// TwinCAT 3 PLC project plc_application1
// ProgramVersion: 3.1.4022.7
// libraries:
//   Tc2_Standard, * (Beckhoff Automation GmbH)
//   Tc2_System, * (Beckhoff Automation GmbH)
//   Tc3_Module, * (Beckhoff Automation GmbH)
// project tree:
//   DUTs/ DUT_1.TcDUT
//   GVLs/ GVL.TcGVL, GVL_1.TcGVL
//   / PlcTask.TcTTO
//   POUs/ MAIN.TcPOU, POU.TcPOU
// real-time tasks:
//   TASK PlcTask: cycle T#10ms, priority 20, ADS port 350
// I/O:
//   DEVICE Device 1 (EtherCAT), AmsNetId 10.1.1.164.2.1

CONFIGURATION plc_application1
    RESOURCE PLC ON TwinCAT3
        TASK PlcTask(INTERVAL := T#10ms, PRIORITY := 20);
        PROGRAM MAIN WITH PlcTask : MAIN;
    END_RESOURCE
END_CONFIGURATION

// ---- DUTs/DUT_1.TcDUT
TYPE DUT_1 :
STRUCT
END_STRUCT
END_TYPE

// ---- GVLs/GVL.TcGVL
{attribute 'qualified_only'}
VAR_GLOBAL
	newTrunks:BOOL;
END_VAR

// ---- GVLs/GVL_1.TcGVL
{attribute 'qualified_only'}
VAR_GLOBAL
		myInt1:INT; (*my var*)
		efhehfi:INT;
		bYAwVar1:BOOL;
		bPickupSensorA:BOOL;
		newVar1:BOOL;
END_VAR

// ---- POUs/MAIN.TcPOU
PROGRAM MAIN
VAR
	hello:BOOL;
	newVar:INT;
	newone:INT;
	nextone:REAL;
	thisisnotInGits_1:REAL;
END_VAR

END_PROGRAM

// ---- POUs/POU.TcPOU
PROGRAM POU
VAR
END_VAR

GVL_1.bYAwVar1:=TRUE;
IF GVL_1.bYAwVar1 THEN
	GVL_1.myInt1:=1;
END_IF

END_PROGRAM
